INTERFACE I_UserDefinedDatatype EXTENDS I_Datatype

PROPERTY PUBLIC Identifier : T_MAXSTRING
GET
END_GET
END_PROPERTY

END_INTERFACE

(* stored: Version 1.1.0.1, ProductVersion 3.1.4024.12
   Itf I_UserDefinedDatatype: Id {c82e94ca-21e4-049b-0a0b-1b0ff127cc32}
   Property Identifier: Id {683c0489-55b3-0103-3b9b-19dd7c7cb00d}
   Get Get: Id {68f3d1a2-0b09-06a4-3b18-fd402adbf535} *)
